(* 
| :Description: This function block use for Contactor active by digital output,
| Use NO contact feedback(Digital Input) to just see, not affect the state control like "FB_contactorFBNO"
*)
FUNCTION_BLOCK FB_ContactorNonFB_Flex EXTENDS FB_ContactorNonFB
VAR
	piNO 		: FB_DigitalInputExt;
END_VAR

SUPER^();

METHOD MR_FirstCycle : BOOL
VAR_INPUT
	sName 							: STRING;
	sCoilModuleType					: STRING;
	sCoilPortID						: STRING;
	sNOModuleType					: STRING;
	sNOPortID						: STRING;
	tGoActiveTimeout				: TIME;
	tDelay							: TIME;
END_VAR
piNO.EnableTimeout := TRUE;
THIS^.sName := sName;								
THIS^.piNO.MR_FirstCycleEx(
	sName := CONCAT(sName,':NO'),
	sModuleType := sNOModuleType,
	sPortID	:= sNOPortID,
	bEnableTimeout := TRUE,
	tDefaultTimeout	:= tGoActiveTimeout
);
THIS^.poCoil.MR_FirstCycle(
	sName := CONCAT(sName,':Coil'),
	sModuleType := sCoilModuleType,
	sPortID := sCoilPortID
);
END_METHOD

PROPERTY Ref_piNO : reference to  FB_DigitalInput
GET
ref_piNO ref= THIS^.piNO;
END_GET
END_PROPERTY

END_FUNCTION_BLOCK

(* stored: Version 1.1.0.1, ProductVersion 3.1.4024.12
   POU FB_ContactorNonFB_Flex: Id {cd50ce4f-283c-434e-8b9d-f759d9bf84f3}, SpecialFunc None
   Method MR_FirstCycle: Id {dbd353e4-ac60-4183-be19-cfe7c161068c}
   Property Ref_piNO: Id {b736aa4e-127a-4cb6-96e1-972eca122214}
   Get Get: Id {244cc720-5090-4e22-be0d-1c653cfa97de} *)
